// TIA Portal V15.1 export
// export: Created 2024-05-17T05:38:29.8172485Z, ExportSetting WithDefaults, DisplayName Totally Integrated Automation Portal, DisplayVersion V15.1 Update 5, DisplayName TIA Portal Openness, DisplayVersion V15.1 Update 5, DisplayName SINAMICS Startdrive Advanced, DisplayVersion V15.1, DisplayName G130, G150, S120, S150, SINAMICS MV, S210, DisplayVersion V15.1, DisplayName G110M, G120, G120C, G120D, G120P, DisplayVersion V15.1, DisplayName STEP 7 Professional, DisplayVersion V15.1 Update 5, DisplayName STEP 7 Safety, DisplayVersion V15.1, DisplayName WinCC Professional, DisplayVersion V15.1 Update 5, DisplayName SIMATIC Visualization Architect, DisplayVersion V15.1
FUNCTION_BLOCK "LPNIODiagS7-1500"   // FB2205, SCL
TITLE = PN_IO for HMI
{ S7_Optimized_Access := 'TRUE' }
AUTHOR : VCC
FAMILY : PNIODiag
VERSION : 0.0.0.0
// apette18,PADA
// stored: AutoNumber false, IsIECCheckEnabled true, IsRetainMemResEnabled true, MemoryReserve 200, RetainMemoryReserve 0, SetENOAutomatically True, UDAEnableTagReadback false
   VAR_INPUT
      I_HWIOSYSTEM { ExternalAccessible := 'False'; ExternalVisible := 'False'; ExternalWritable := 'False'} : HW_IOSYSTEM;   // HW ID ProfiNet System
      I_PLCIOSYSTEM { ExternalAccessible := 'False'; ExternalVisible := 'False'; ExternalWritable := 'False'} : HW_INTERFACE;   // HW ID ProfiNet System PLC Port 1
      I_LastDeviceNumber { ExternalAccessible := 'False'; ExternalVisible := 'False'; ExternalWritable := 'False'} : Int;   // Last Device of ProfiNet System
   END_VAR
   VAR_OUTPUT
      O_LastDeviceNumber { ExternalAccessible := 'False'; ExternalVisible := 'False'; ExternalWritable := 'False'} : Int;   // Last Device of ProfiNet System
   END_VAR
   VAR_IN_OUT
      IO_DeviceExist : Array[0..255] of Bool;   // IO devices exist
      IO_HWIdentifier : Array[0..255] of UInt;   // HW Device
      IO_PNIODIAG_Global : "H_PNIODiagS7-1500";
   END_VAR
   VAR
      PNDeviceConfigured { ExternalAccessible := 'False'; ExternalVisible := 'False'; ExternalWritable := 'False'} : Array[0..255] of Bool;   // IO devices are configured
      PNDeviceExist { ExternalAccessible := 'False'; ExternalVisible := 'False'; ExternalWritable := 'False'} : Array[0..255] of Bool;   // IO devices are faulty
      PNDeviceFaulty { ExternalAccessible := 'False'; ExternalVisible := 'False'; ExternalWritable := 'False'} : Array[0..255] of Bool;   // IO devices are faulty
      PNDeviceDisabled { ExternalAccessible := 'False'; ExternalVisible := 'False'; ExternalWritable := 'False'} : Array[0..255] of Bool;   // IO devices are disabled
      PNDeviceServiceReq { ExternalAccessible := 'False'; ExternalVisible := 'False'; ExternalWritable := 'False'} : Array[0..255] of Bool;   // IO devices for which a problem has occurred
      Edge { ExternalAccessible := 'False'; ExternalVisible := 'False'; ExternalWritable := 'False'} : Bool;   // Temp
      GeoAdress { ExternalAccessible := 'False'; ExternalVisible := 'False'; ExternalWritable := 'False'; S7_SetPoint := 'True'} : GEOADDR;   // Int Function
      _ReadIP { ExternalAccessible := 'False'; ExternalVisible := 'False'; ExternalWritable := 'False'; S7_SetPoint := 'True'} : "LPNIODiagReadIPS7-1500";   // FB
      TimerResetPNStatus { ExternalAccessible := 'False'; ExternalVisible := 'False'; ExternalWritable := 'False'; S7_SetPoint := 'True'} : TP_TIME;   // Timer
   END_VAR
   VAR_TEMP
      No1 : Int;   // Temp
      ReturnMode1 : Int;   // Temp
      ReturnMode2 : Int;   // Temp
      ReturnMode3 : Int;   // Temp
      ReturnMode4 : Int;   // Temp
      ReturnMode5 : Int;   // Temp
      ReturnGeo : Int;   // Temp
      ReturnActPNIO : Int;   // Temp
   END_VAR
   // GeoAdress.HWTYPE := 2;
   // GeoAdress.AREA := 1;
   // GeoAdress.IOSYSTEM := 100;
BEGIN

   //**** 1 - Inputs **** Activate Scan
   IF "TRUE" THEN
       #ReturnMode1 := DeviceStates(LADDR := #I_HWIOSYSTEM, MODE := 1, STATE := #PNDeviceConfigured); //1:IO devices are configured
       #ReturnMode2 := DeviceStates(LADDR := #I_HWIOSYSTEM, MODE := 2, STATE := #PNDeviceFaulty); //2: IO devices are faulty   
       #ReturnMode3 := DeviceStates(LADDR := #I_HWIOSYSTEM, MODE := 3, STATE := #PNDeviceDisabled); //3: IO devices are disabled
       #ReturnMode4 := DeviceStates(LADDR := #I_HWIOSYSTEM, MODE := 4, STATE := #PNDeviceExist); //4: IO devices exist
       #ReturnMode5 := DeviceStates(LADDR := #I_HWIOSYSTEM, MODE := 5, STATE := #PNDeviceServiceReq); //5: IO devices for which a problem has occurred    
   END_IF;

   //**** 2.2 - Alarms - Alarm Generation **** Reset Alarm and Warning
   #IO_PNIODIAG_Global.GlobStat_DeviceFaulty := FALSE;
   #IO_PNIODIAG_Global.GlobStat_DeviceDisabled := FALSE;
   #IO_PNIODIAG_Global.GlobStat_DeviceServiceReq := FALSE;

   //**** 4.4 - Machine status - Calculated  **** Set Status color on the HMI
   FOR #No1 := 1 TO #I_LastDeviceNumber DO
       IF #PNDeviceConfigured[#No1] THEN

           //Get HW_DEVICE number from all PN devices that are aviable on the PROFINET
           #GeoAdress.AREA := 1;
           #GeoAdress.HWTYPE := 2;
           #GeoAdress.STATION := INT_TO_UINT(#No1);
           #ReturnGeo := GEO2LOG(GEOADDR := #GeoAdress, LADDR => #IO_HWIdentifier[#No1]);

           //Check If IO Devices Are Faulty
           IF #PNDeviceFaulty[#No1] THEN
               #IO_PNIODIAG_Global.DeviceColor[#No1]:= 1; //red
               #IO_PNIODIAG_Global.DeviceFaulty[#No1] := True;
               #IO_PNIODIAG_Global.DeviceDisabled[#No1] := False;
               #IO_PNIODIAG_Global.DeviceServiceReq[#No1] := False;
               #IO_PNIODIAG_Global.GlobStat_DeviceFaulty := True;
               #IO_PNIODIAG_Global.GlobStat_DeviceDisabled := False;
               #IO_PNIODIAG_Global.GlobStat_DeviceServiceReq := False;

               //Check If  Maintenance Demand Or Service Request Is Active   
           ELSIF #PNDeviceServiceReq[#No1] = TRUE THEN
               #IO_PNIODIAG_Global.DeviceColor[#No1] := 4; //yellow
               #IO_PNIODIAG_Global.DeviceServiceReq[#No1] := True;
               #IO_PNIODIAG_Global.GlobStat_DeviceServiceReq := True;

               //Check if IO Devices Are disabled
           ELSIF #PNDeviceDisabled[#No1] = TRUE THEN
               #IO_PNIODIAG_Global.DeviceColor[#No1] := 2; //blue
               #IO_PNIODIAG_Global.DeviceDisabled[#No1] := True;
               #IO_PNIODIAG_Global.DeviceFaulty[#No1] := False;
               #IO_PNIODIAG_Global.GlobStat_DeviceFaulty := False;
               #IO_PNIODIAG_Global.GlobStat_DeviceDisabled := True;

               //Check If IO Devices Are Existing Without Error/Fault
           ELSIF #PNDeviceExist[#No1] = TRUE THEN
               #IO_PNIODIAG_Global.DeviceColor[#No1] := 3; //green
           END_IF;
       END_IF;
   END_FOR;


   //**** 4.4 - Machine status - Calculated  **** Get IP Address of PLC
   #_ReadIP(I_ReqIN := "TRUE",
            I_HWID := #I_PLCIOSYSTEM);


   //**** 4.4 - Machine status - Calculated  **** Reset the status from the HMI
   IF #IO_PNIODIAG_Global.HMICmd_ResetPNStatus AND NOT #Edge THEN
       #Edge := TRUE;
       FOR #No1 := 1 TO #I_LastDeviceNumber DO
           #IO_PNIODIAG_Global.DeviceFaulty[#No1] := FALSE;
           #IO_PNIODIAG_Global.DeviceDisabled[#No1] := FALSE;
           #IO_PNIODIAG_Global.DeviceServiceReq[#No1] := FALSE;
           #IO_PNIODIAG_Global.GlobStat_DeviceFaulty := FALSE;
           #IO_PNIODIAG_Global.GlobStat_DeviceDisabled := FALSE;
           #IO_PNIODIAG_Global.GlobStat_DeviceServiceReq := FALSE;
       END_FOR;
       #Edge := FALSE;
   END_IF;
   #TimerResetPNStatus(IN:=#IO_PNIODIAG_Global.HMICmd_ResetPNStatus,
                       PT:=T#500ms);
   //IF #TimerResetPNStatus.Q THEN
   //    #IO_PNIODIAG_Global.HMICmd_ResetPNStatus := False;
   //END_IF;


   //**** 4.4 - Machine status - Calculated  **** Activate or Deactivate PN Devices
   #ReturnActPNIO := D_ACT_DP(REQ := #IO_PNIODIAG_Global.HMICmd_ActivateDeactivate, MODE :=#IO_PNIODIAG_Global.PNMode, LADDR := #IO_HWIdentifier[ #IO_PNIODIAG_Global.DeviceNumber], BUSY => #IO_PNIODIAG_Global.ActivateDeactivateBusy);
   #IO_PNIODIAG_Global.HMICmd_ActivateDeactivate := FALSE;


   // **** 4.6 - Machine status - Indication ****  Animation
   #IO_PNIODIAG_Global.IPAddressPLC[0]:= #_ReadIP.O_IPParam.IPAddress[0];
   #IO_PNIODIAG_Global.IPAddressPLC[1] := #_ReadIP.O_IPParam.IPAddress[1];
   #IO_PNIODIAG_Global.IPAddressPLC[2] := #_ReadIP.O_IPParam.IPAddress[2];
   #IO_PNIODIAG_Global.IPAddressPLC[3] := #_ReadIP.O_IPParam.IPAddress[3];

   #IO_PNIODIAG_Global.DeviceExist := #PNDeviceExist;
   #IO_DeviceExist := #PNDeviceExist;

   #O_LastDeviceNumber := #I_LastDeviceNumber;
END_FUNCTION_BLOCK
